{attribute 'qualified_only'}
VAR_GLOBAL
END_VAR

(* stored: Version 1.1.0.1, ProductVersion 3.1.4022.7
   GVL GVL_04_Auto_All: Id {48b88134-d685-4aa8-acc8-7eb4e36572d5} *)
